Omron CX-Programmer project NewProject (CX-Programmer 9.75)

# PLC NewPLC1: CP1H XA

## Global symbols (name address type ; comment)
0.00 BOOL  ; PB Start
0.01 BOOL  ; PB Stop
100.00 BOOL  ; Internal Relay
100.01 BOOL  ; MERAH S1
100.02 BOOL  ; KUNING S1
100.03 BOOL  ; HIJAU S1
100.04 BOOL  ; MERAH S2
100.05 BOOL  ; KUNING S2
100.06 BOOL  ; HIJAU S2
100.07 BOOL  ; MERAH S3
100.08 BOOL  ; KUNING S3
100.09 BOOL  ; HIJAU S3
100.10 BOOL  ; MERAH S4
100.11 BOOL  ; KUNING S4
100.12 BOOL  ; HIJAU S4
100.13 BOOL  ; PB Stop
100.14 BOOL  ; 5dtk
100.15 BOOL  ; 2
101.00 BOOL  ; KUNING S3
101.01 BOOL  ; HIJAU S3
101.02 BOOL  ; MERAH S4
101.03 BOOL  ; KUNING S4
101.04 BOOL  ; HIJAU S4
11.00 BOOL  ; normal
11.01 BOOL  ; Lampu kedip
1.00 BOOL  ; Kuning 5 dtk
A351 CHANNEL  ; EXTRA
A352 CHANNEL  ; jumat
A354 CHANNEL  ; S - J
D100 CHANNEL  ; JAM 2
D110 CHANNEL  ; JAM 23
D120 CHANNEL  ; JAM 6
D130 CHANNEL  ; JAM 8
T0000 BOOL  ; Merah 20
T0002 BOOL  ; T HIJAU 1
T0003 BOOL  ; T KUNING 1
T0004 BOOL  ; T MERAH 1
T0005 BOOL  ; T HIJAU 2
T0006 BOOL  ; T KUNING 2
T0007 BOOL  ; T MERAH 2
T0008 BOOL  ; T HIJAU 3
T0009 BOOL  ; T KUNING 3
T0010 BOOL  ; T MERAH 3
T0011 BOOL  ; T HIJAU 4
T0012 BOOL  ; T KUNING 4
T0013 BOOL  ; T MERAH 4
W10.00 BOOL  ; IR
W10.02 BOOL  ; hari s - j
W10.03 BOOL  ; 6 - 8
W11.00 BOOL  ; program awal
W11.01 BOOL  ; MERAH S1
W11.02 BOOL  ; KUNING S1
W11.03 BOOL  ; HIJAU S1
W11.04 BOOL  ; MERAH S2
W11.05 BOOL  ; KUNING S2
W11.06 BOOL  ; HIJAU S2
W11.07 BOOL  ; MERAH S3
W11.08 BOOL  ; KUNING S3
W11.09 BOOL  ; HIJAU S3
W11.10 BOOL  ; MERAH S4
W11.11 BOOL  ; KUNING S4
W11.12 BOOL  ; HIJAU S4
W11.13 BOOL  ; K KEDIP
W12.01 BOOL  ; gab kuning 1
W12.02 BOOL  ; gab kuning 2
W12.03 BOOL  ; gab kuning 3
W12.04 BOOL  ; gab kuning 4
W12.12 BOOL  ; HIJAU S4

## Program NewProgram1 (cyclic task 0)
Local symbols
DT UINT
R4 BOOL

### Section Section1

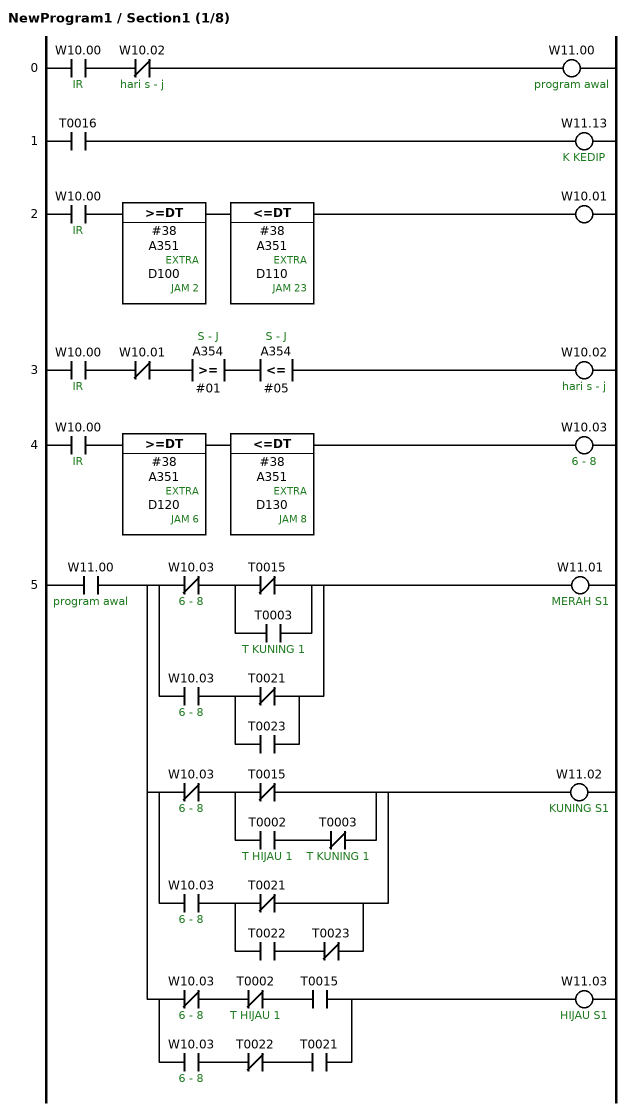
; rung 0
LD W10.00  ; IR
ANDNOT W10.02  ; hari s - j
OUT W11.00  ; program awal
; rung 1
LD T0016
OUT W11.13  ; K KEDIP
; rung 2
LD W10.00  ; IR
AND>=DT(346) #38 A351 D100  ; EXTRA, JAM 2
AND<=DT(344) #38 A351 D110  ; EXTRA, JAM 23
OUT W10.01
; rung 3
LD W10.00  ; IR
ANDNOT W10.01
AND>=(325) A354 #01  ; S - J
AND<=(315) A354 #05  ; S - J
OUT W10.02  ; hari s - j
; rung 4
LD W10.00  ; IR
AND>=DT(346) #38 A351 D120  ; EXTRA, JAM 6
AND<=DT(344) #38 A351 D130  ; EXTRA, JAM 8
OUT W10.03  ; 6 - 8
; rung 5
LD W11.00  ; program awal
OUT TR0
LDNOT W10.03  ; 6 - 8
LDNOT T0015
OR T0003  ; T KUNING 1
ANDLD
LD W10.03  ; 6 - 8
LDNOT T0021
OR T0023
ANDLD
ORLD
ANDLD
OUT W11.01  ; MERAH S1
LD TR0
LDNOT W10.03  ; 6 - 8
LDNOT T0015
LD T0002  ; T HIJAU 1
ANDNOT T0003  ; T KUNING 1
ORLD
ANDLD
LD W10.03  ; 6 - 8
LDNOT T0021
LD T0022
ANDNOT T0023
ORLD
ANDLD
ORLD
ANDLD
OUT W11.02  ; KUNING S1
LD TR0
LDNOT W10.03  ; 6 - 8
ANDNOT T0002  ; T HIJAU 1
AND T0015
LD W10.03  ; 6 - 8
ANDNOT T0022
AND T0021
ORLD
ANDLD
OUT W11.03  ; HIJAU S1

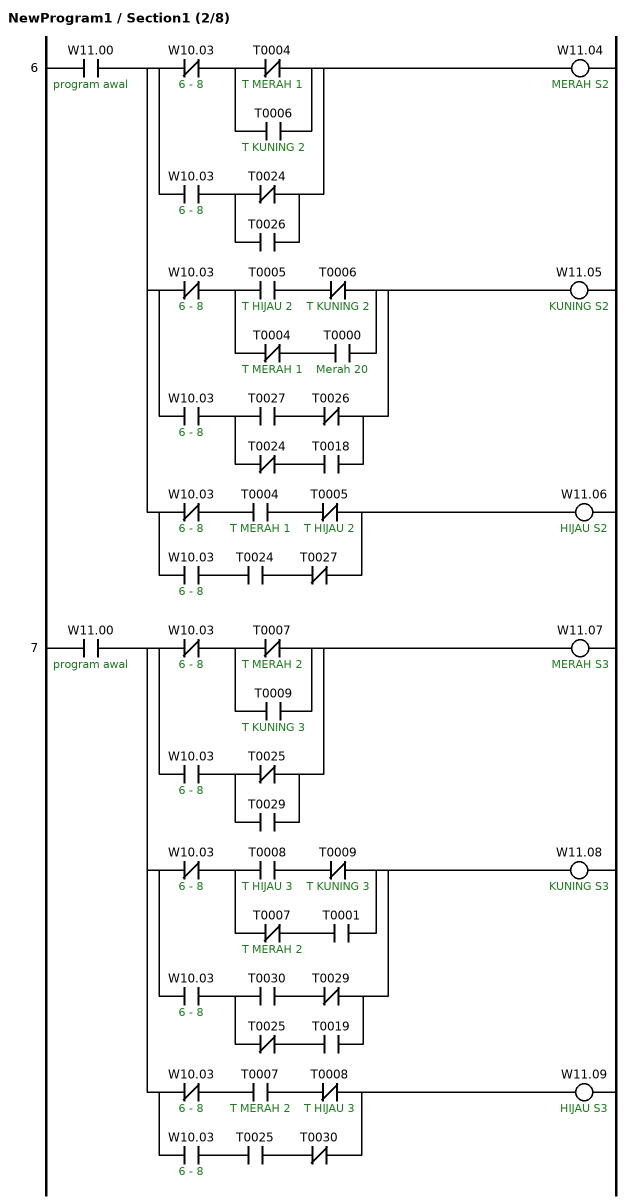
; rung 6
LD W11.00  ; program awal
OUT TR0
LDNOT W10.03  ; 6 - 8
LDNOT T0004  ; T MERAH 1
OR T0006  ; T KUNING 2
ANDLD
LD W10.03  ; 6 - 8
LDNOT T0024
OR T0026
ANDLD
ORLD
ANDLD
OUT W11.04  ; MERAH S2
LD TR0
LDNOT W10.03  ; 6 - 8
LD T0005  ; T HIJAU 2
ANDNOT T0006  ; T KUNING 2
LDNOT T0004  ; T MERAH 1
AND T0000  ; Merah 20
ORLD
ANDLD
LD W10.03  ; 6 - 8
LD T0027
ANDNOT T0026
LDNOT T0024
AND T0018
ORLD
ANDLD
ORLD
ANDLD
OUT W11.05  ; KUNING S2
LD TR0
LDNOT W10.03  ; 6 - 8
AND T0004  ; T MERAH 1
ANDNOT T0005  ; T HIJAU 2
LD W10.03  ; 6 - 8
AND T0024
ANDNOT T0027
ORLD
ANDLD
OUT W11.06  ; HIJAU S2
; rung 7
LD W11.00  ; program awal
OUT TR0
LDNOT W10.03  ; 6 - 8
LDNOT T0007  ; T MERAH 2
OR T0009  ; T KUNING 3
ANDLD
LD W10.03  ; 6 - 8
LDNOT T0025
OR T0029
ANDLD
ORLD
ANDLD
OUT W11.07  ; MERAH S3
LD TR0
LDNOT W10.03  ; 6 - 8
LD T0008  ; T HIJAU 3
ANDNOT T0009  ; T KUNING 3
LDNOT T0007  ; T MERAH 2
AND T0001
ORLD
ANDLD
LD W10.03  ; 6 - 8
LD T0030
ANDNOT T0029
LDNOT T0025
AND T0019
ORLD
ANDLD
ORLD
ANDLD
OUT W11.08  ; KUNING S3
LD TR0
LDNOT W10.03  ; 6 - 8
AND T0007  ; T MERAH 2
ANDNOT T0008  ; T HIJAU 3
LD W10.03  ; 6 - 8
AND T0025
ANDNOT T0030
ORLD
ANDLD
OUT W11.09  ; HIJAU S3

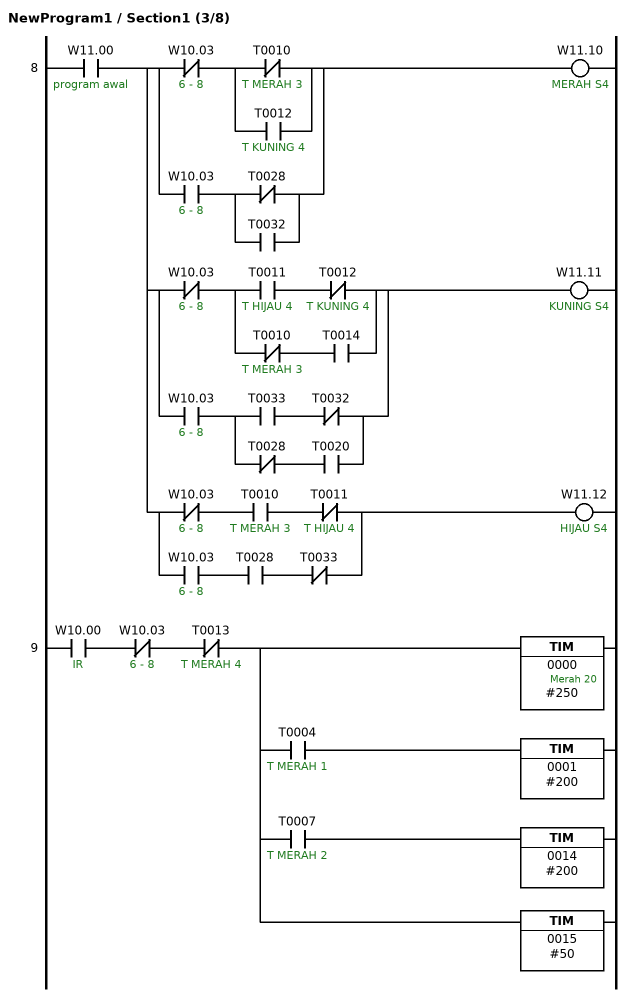
; rung 8
LD W11.00  ; program awal
OUT TR0
LDNOT W10.03  ; 6 - 8
LDNOT T0010  ; T MERAH 3
OR T0012  ; T KUNING 4
ANDLD
LD W10.03  ; 6 - 8
LDNOT T0028
OR T0032
ANDLD
ORLD
ANDLD
OUT W11.10  ; MERAH S4
LD TR0
LDNOT W10.03  ; 6 - 8
LD T0011  ; T HIJAU 4
ANDNOT T0012  ; T KUNING 4
LDNOT T0010  ; T MERAH 3
AND T0014
ORLD
ANDLD
LD W10.03  ; 6 - 8
LD T0033
ANDNOT T0032
LDNOT T0028
AND T0020
ORLD
ANDLD
ORLD
ANDLD
OUT W11.11  ; KUNING S4
LD TR0
LDNOT W10.03  ; 6 - 8
AND T0010  ; T MERAH 3
ANDNOT T0011  ; T HIJAU 4
LD W10.03  ; 6 - 8
AND T0028
ANDNOT T0033
ORLD
ANDLD
OUT W11.12  ; HIJAU S4
; rung 9
LD W10.00  ; IR
ANDNOT W10.03  ; 6 - 8
ANDNOT T0013  ; T MERAH 4
OUT TR0
TIM 0000 #250  ; Merah 20
AND T0004  ; T MERAH 1
TIM 0001 #200
LD TR0
AND T0007  ; T MERAH 2
TIM 0014 #200
LD TR0
TIM 0015 #50

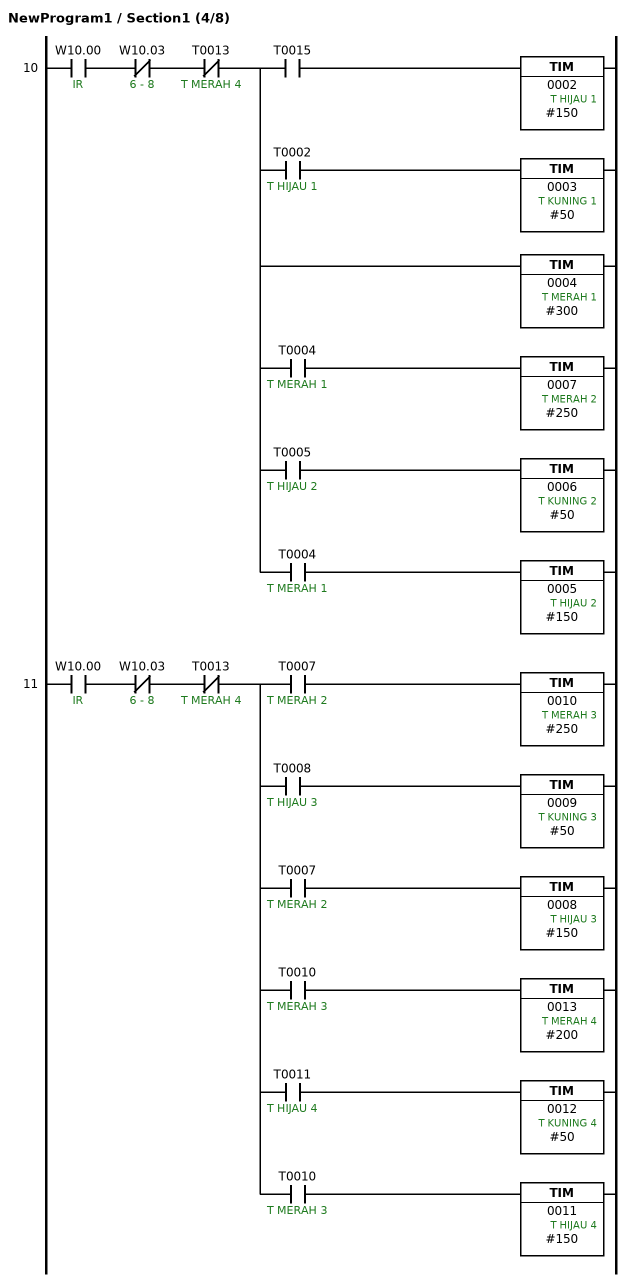
; rung 10
LD W10.00  ; IR
ANDNOT W10.03  ; 6 - 8
ANDNOT T0013  ; T MERAH 4
OUT TR0
AND T0015
TIM 0002 #150  ; T HIJAU 1
LD TR0
AND T0002  ; T HIJAU 1
TIM 0003 #50  ; T KUNING 1
LD TR0
TIM 0004 #300  ; T MERAH 1
AND T0004  ; T MERAH 1
TIM 0007 #250  ; T MERAH 2
LD TR0
AND T0005  ; T HIJAU 2
TIM 0006 #50  ; T KUNING 2
LD TR0
AND T0004  ; T MERAH 1
TIM 0005 #150  ; T HIJAU 2
; rung 11
LD W10.00  ; IR
ANDNOT W10.03  ; 6 - 8
ANDNOT T0013  ; T MERAH 4
OUT TR0
AND T0007  ; T MERAH 2
TIM 0010 #250  ; T MERAH 3
LD TR0
AND T0008  ; T HIJAU 3
TIM 0009 #50  ; T KUNING 3
LD TR0
AND T0007  ; T MERAH 2
TIM 0008 #150  ; T HIJAU 3
LD TR0
AND T0010  ; T MERAH 3
TIM 0013 #200  ; T MERAH 4
LD TR0
AND T0011  ; T HIJAU 4
TIM 0012 #50  ; T KUNING 4
LD TR0
AND T0010  ; T MERAH 3
TIM 0011 #150  ; T HIJAU 4

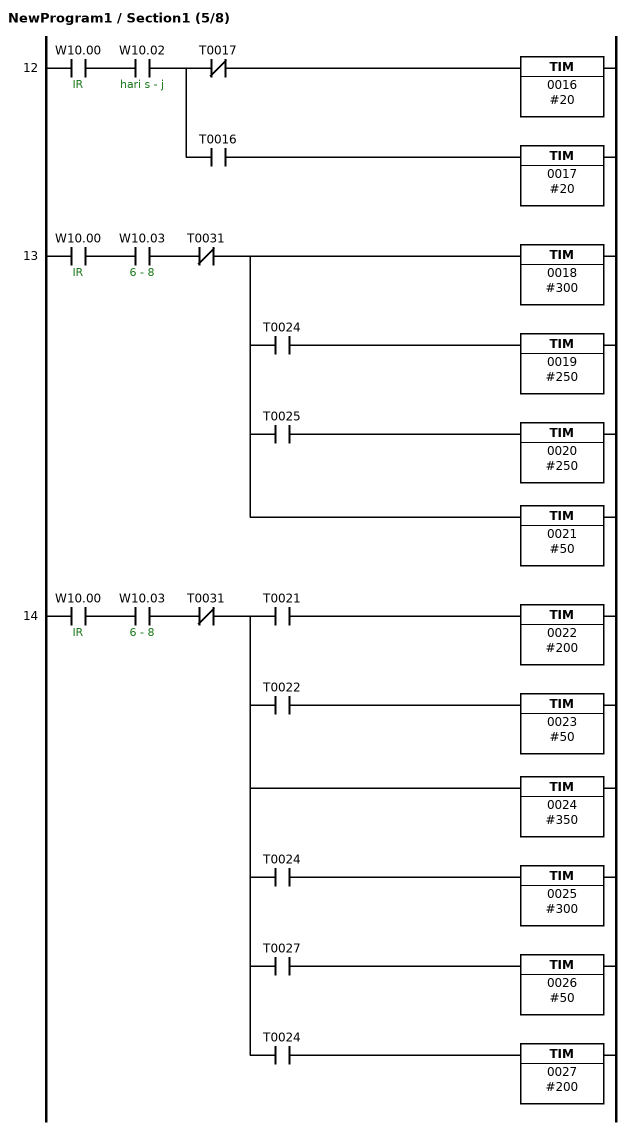
; rung 12
LD W10.00  ; IR
AND W10.02  ; hari s - j
OUT TR0
ANDNOT T0017
TIM 0016 #20
LD TR0
AND T0016
TIM 0017 #20
; rung 13
LD W10.00  ; IR
AND W10.03  ; 6 - 8
ANDNOT T0031
OUT TR0
TIM 0018 #300
AND T0024
TIM 0019 #250
LD TR0
AND T0025
TIM 0020 #250
LD TR0
TIM 0021 #50
; rung 14
LD W10.00  ; IR
AND W10.03  ; 6 - 8
ANDNOT T0031
OUT TR0
AND T0021
TIM 0022 #200
LD TR0
AND T0022
TIM 0023 #50
LD TR0
TIM 0024 #350
AND T0024
TIM 0025 #300
LD TR0
AND T0027
TIM 0026 #50
LD TR0
AND T0024
TIM 0027 #200

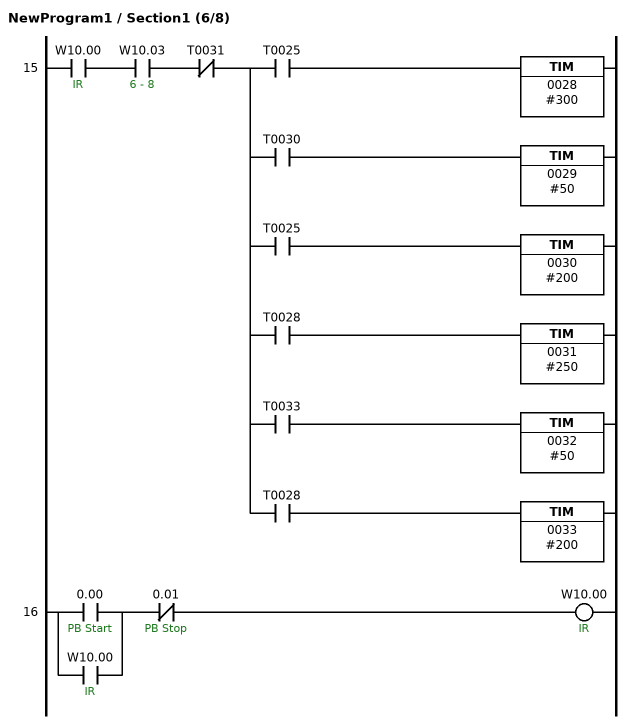
; rung 15
LD W10.00  ; IR
AND W10.03  ; 6 - 8
ANDNOT T0031
OUT TR0
AND T0025
TIM 0028 #300
LD TR0
AND T0030
TIM 0029 #50
LD TR0
AND T0025
TIM 0030 #200
LD TR0
AND T0028
TIM 0031 #250
LD TR0
AND T0033
TIM 0032 #50
LD TR0
AND T0028
TIM 0033 #200
; rung 16
LD 0.00  ; PB Start
OR W10.00  ; IR
ANDNOT 0.01  ; PB Stop
OUT W10.00  ; IR

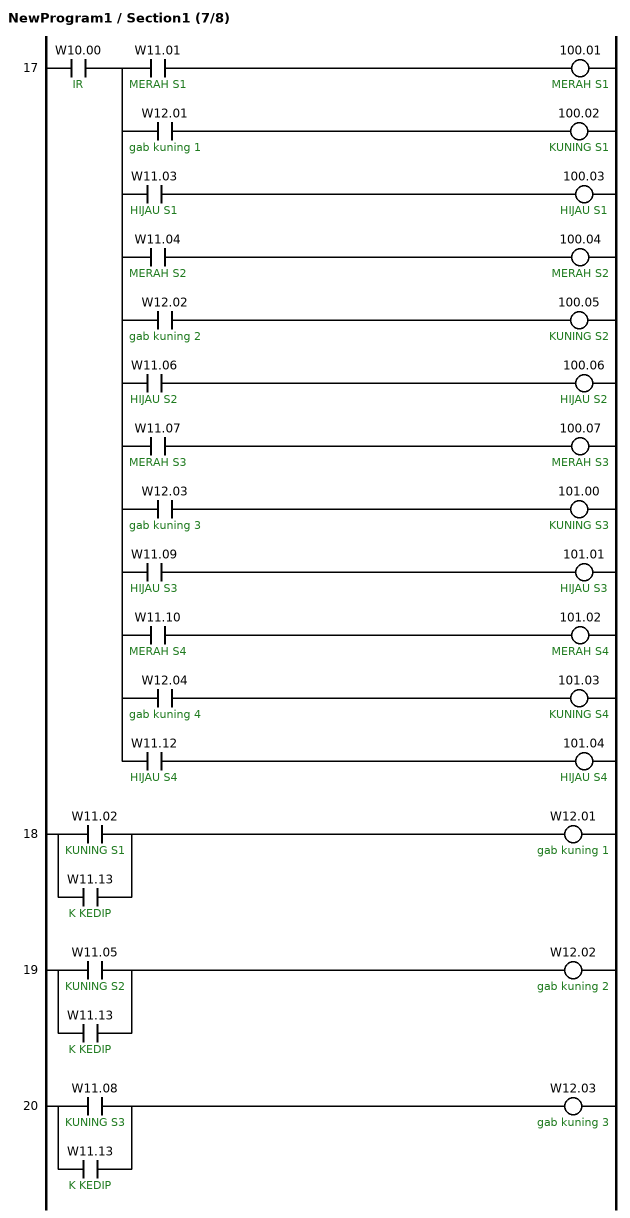
; rung 17
LD W10.00  ; IR
OUT TR0
AND W11.01  ; MERAH S1
OUT 100.01  ; MERAH S1
LD TR0
AND W12.01  ; gab kuning 1
OUT 100.02  ; KUNING S1
LD TR0
AND W11.03  ; HIJAU S1
OUT 100.03  ; HIJAU S1
LD TR0
AND W11.04  ; MERAH S2
OUT 100.04  ; MERAH S2
LD TR0
AND W12.02  ; gab kuning 2
OUT 100.05  ; KUNING S2
LD TR0
AND W11.06  ; HIJAU S2
OUT 100.06  ; HIJAU S2
LD TR0
AND W11.07  ; MERAH S3
OUT 100.07  ; MERAH S3
LD TR0
AND W12.03  ; gab kuning 3
OUT 101.00  ; KUNING S3
LD TR0
AND W11.09  ; HIJAU S3
OUT 101.01  ; HIJAU S3
LD TR0
AND W11.10  ; MERAH S4
OUT 101.02  ; MERAH S4
LD TR0
AND W12.04  ; gab kuning 4
OUT 101.03  ; KUNING S4
LD TR0
AND W11.12  ; HIJAU S4
OUT 101.04  ; HIJAU S4
; rung 18
LD W11.02  ; KUNING S1
OR W11.13  ; K KEDIP
OUT W12.01  ; gab kuning 1
; rung 19
LD W11.05  ; KUNING S2
OR W11.13  ; K KEDIP
OUT W12.02  ; gab kuning 2
; rung 20
LD W11.08  ; KUNING S3
OR W11.13  ; K KEDIP
OUT W12.03  ; gab kuning 3

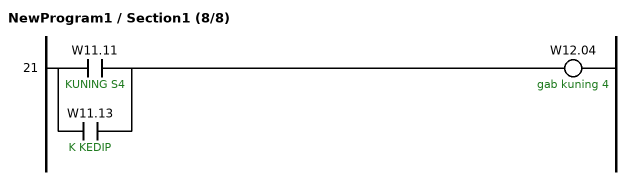
; rung 21
LD W11.11  ; KUNING S4
OR W11.13  ; K KEDIP
OUT W12.04  ; gab kuning 4

### Section END
; rung 0
END(001)